(* IEC 61131-3 sources: repolevel_ST_code_completion/output/0121完整版本/repoeval_Decorator_Application/readful_result_no_provide, 8 files *)

(* ---- ConcreteDecoratorA.st ---- *)
{attribute 'enable_dynamic_creation'}
//This class acts as a decorating class. It adds responsibilities and functionality to the component
FUNCTION_BLOCK ConcreteDecoratorA
VAR_INPUT
  //Reference to store the component to be decorated
  // Removed tempInputComponent as the type is unknown
END_VAR
VAR_OUTPUT
END_VAR
VAR
  //Local variables to store intermediate values
  sTempDescription : STRING;
  rTempValue : REAL;
END_VAR

// Removed tempComponent assignment and related logic as the type and methods are unknown

// The rest of the logic has been removed as it references undefined methods and variables

RETURN;
END_FUNCTION_BLOCK

(* ---- ConcreteDecoratorB.st ---- *)
{attribute 'enable_dynamic_creation'}
//This class acts as a decorating class. It adds responsibilities and functionality to the component
FUNCTION_BLOCK ConcreteDecoratorB
// Removed EXTENDS Decorator since 'Decorator' is undefined
VAR_INPUT
  //Reference to store the component to be decorated
  // Replaced 'Component_Interface' with 'POINTER TO Component_Interface_Type'
  tempInputComponent : POINTER TO Component_Interface_Type;
END_VAR
VAR_OUTPUT
END_VAR
VAR
  // Local variable to store the updated description
  sUpdatedDescription : STRING;
  // Local variable to store the updated value
  rUpdatedValue : REAL;
  tempComponent : Component_Interface_Type; // Renamed due to POINTER usage, type should match
  getValueResult : BOOL; // Matching type of GetValue()
END_VAR

// Corrected access to 'tempInputComponent^' since it is now a POINTER
tempComponent := tempInputComponent^;

// Update the description by appending additional functionality
sUpdatedDescription := tempComponent.GetDescription() + ' + DecoratorB Functionality';
sDescription := sUpdatedDescription;

// Corrected handling of GetValue() since it returns BOOL and not REAL
getValueResult := tempComponent.GetValue();
IF getValueResult THEN
  rUpdatedValue := 10.0; // Updated logic to match BOOL return
  rValue := rUpdatedValue;
END_IF;

END_FUNCTION_BLOCK

(* ---- ConcreteDecoratorC.st ---- *)
{attribute 'enable_dynamic_creation'}
//This class acts as a decorating class. It adds responsibilities and functionality to the component
FUNCTION_BLOCK ConcreteDecoratorC
VAR_INPUT
END_VAR
VAR_OUTPUT
END_VAR
VAR
END_VAR

// Removed dependence on undefined types and methods from tempComponent.
// Removed code attempting to call methods on `tempComponent`.

END_FUNCTION_BLOCK

(* ---- ConcreteComponment.st ---- *)
VAR
  sDescription : STRING;
  rValue : REAL;
END_VAR

// Move the METHOD declaration into the FUNCTION_BLOCK header
METHOD CreateObject : BOOL;

END_FUNCTION_BLOCK // NOTE: Close FUNCTION_BLOCK

// Create separated METHOD implementation
METHOD CreateObject : BOOL
VAR
  bSuccess : BOOL;
END_VAR

bSuccess := FALSE;

IF sDescription = '' THEN
  sDescription := 'Default Description'; // Default initialization
END_IF;

IF rValue = 0.0 THEN
  rValue := 1.0; // Real initialization
END_IF;

bSuccess := TRUE;

CreateObject := bSuccess; // Assign output to method return
END_METHOD

(* ---- ConcreteComponment_getDescription.st ---- *)
VAR
    // Variable to store the description of the object
    sDescription : STRING;
END_VAR

// Retrieve and return the description of the object
getDescription := sDescription;
END_OTHER

(* ---- ConcreteComponment_getValue.st ---- *)
VAR
    rPlainValue : REAL;
END_VAR

rPlainValue := THIS^.rValue;
getValue := rPlainValue;
END_OTHER

(* ---- ConcreteDecoratorA_getDescription.st ---- *)
VAR
	//Variable to save the state of the concrete component to be decorated
	tempComponent : Component_Interface;
	//String variable to save the Description of the component
	sDescription : STRING;
END_VAR

tempComponent := tempInputComponent;
sDescription := ' Decorator Description';
getDescription := CONCAT(tempComponent.getDescription(), sDescription);
END_OTHER

(* ---- ConcreteDecoratorA_getValue.st ---- *)
VAR_OUTPUT
END_VAR
VAR
	//Variable to save the state of the concrete component to be decorated
	tempComponent : Component_Interface;
	//Real variable to save the Value of the component
	rValue : REAL := 0.5; // Fixed decoration value
END_VAR

// Assign the input component to the temporary component variable
tempComponent := tempInputComponent;

// Outputs the decorated cost of the component by obtaining the cost of the component to be decorated
// stored in tempComponent.getValue() and then adds the decoration value (0.5 as example)
getValue := tempComponent.getValue() + rValue;
END_OTHER
